// TIA Portal V16 export
// export: Created 2024-12-03T15:41:45.8001006Z, ExportSetting WithReadOnly, DisplayName Totally Integrated Automation Portal, DisplayVersion V16 Update 6, DisplayName TIA Portal Version Control Interface, DisplayVersion V16 Update 2, DisplayName TIA Portal Openness, DisplayVersion V16 Update 6, DisplayName TIA Portal Teamcenter Gateway, DisplayVersion V16, DisplayName SINAMICS Startdrive Advanced, DisplayVersion V16 Update 5, DisplayName SINAMICS Startdrive G130, G150, S120, S150, SINAMICS MV, S210, DisplayVersion V16 Update 5, DisplayName SINAMICS Startdrive G110M, G120, G120C, G120D, G120P, G115D, DisplayVersion V16 Update 5, DisplayName STEP 7 Professional, DisplayVersion V16 Update 6, DisplayName STEP 7 Safety, DisplayVersion V16, DisplayName WinCC Advanced / Unified PC, DisplayVersion V16 Update 6
TYPE "Nord_Shute_Drive_UDT"
// stored: CreationDate 2023-04-19T11:30:38.0051651Z, InterfaceModifiedDate 2023-04-19T12:03:36.128334Z, IsConsistent true, LibraryConformanceStatus The object is library-conformant., ModifiedDate 2023-04-19T12:03:36.128334Z
   STRUCT
      Cmd : Struct   // MotorCommands
         Reset : Bool;
         Auto : Struct
            cmd_move : Bool;
            speed : Real;
         END_STRUCT;
         Manual : Struct
            cmd_move : Bool;
            home : Bool;
            speed : Real;
         END_STRUCT;
         Interlock : Bool;
      END_STRUCT;
      Alarms : Struct
         ServoModeTimedOut_x0 : Bool;   // Motor not on in time
         NotInHome_x1 : Bool;   // Motor not off in time
         HomingTimedout_x2 : Bool;
         ErrorFromDrive_x3 : Bool;   // Error from drive
         CannotStartError_x4 : Bool;   // Cannot start error
         EmergencyStopActive_x5 : Bool;   // Emergency stop is active
         Disconnected_x6 : Bool;   // The device is not connected
         WarningFromDrive_x7 { S7_SetPoint := 'True'} : Bool;   // Warning from drive
         AlarmStatus : Word;   // lsb 0 not on | lsb 1 not off | lsb 2 error from drive | lsb 3 cannot start | 4 emergency stop active | 5 disconnected
      END_STRUCT;
      Status : Struct
         Interlocked : Bool;
         ManualModeActive : Bool;
         ManualCommandsDisabled : Bool;
         running : Bool;
         homed : Bool;
         movement_done : "SmartBooldt";
         in_home : Bool;
         ActualSpeed : Real;
         ActualDirection : Bool;   // 0 right | 1 left
         ReadyToStart : Bool;
         ReadyForOperaiton : Bool;
         PowerOn : Bool;
      END_STRUCT;
      Settings : Struct
         direction : Bool;
      END_STRUCT;
      Zone : Int;
      info : "MotorInfo";
   END_STRUCT;
END_TYPE
